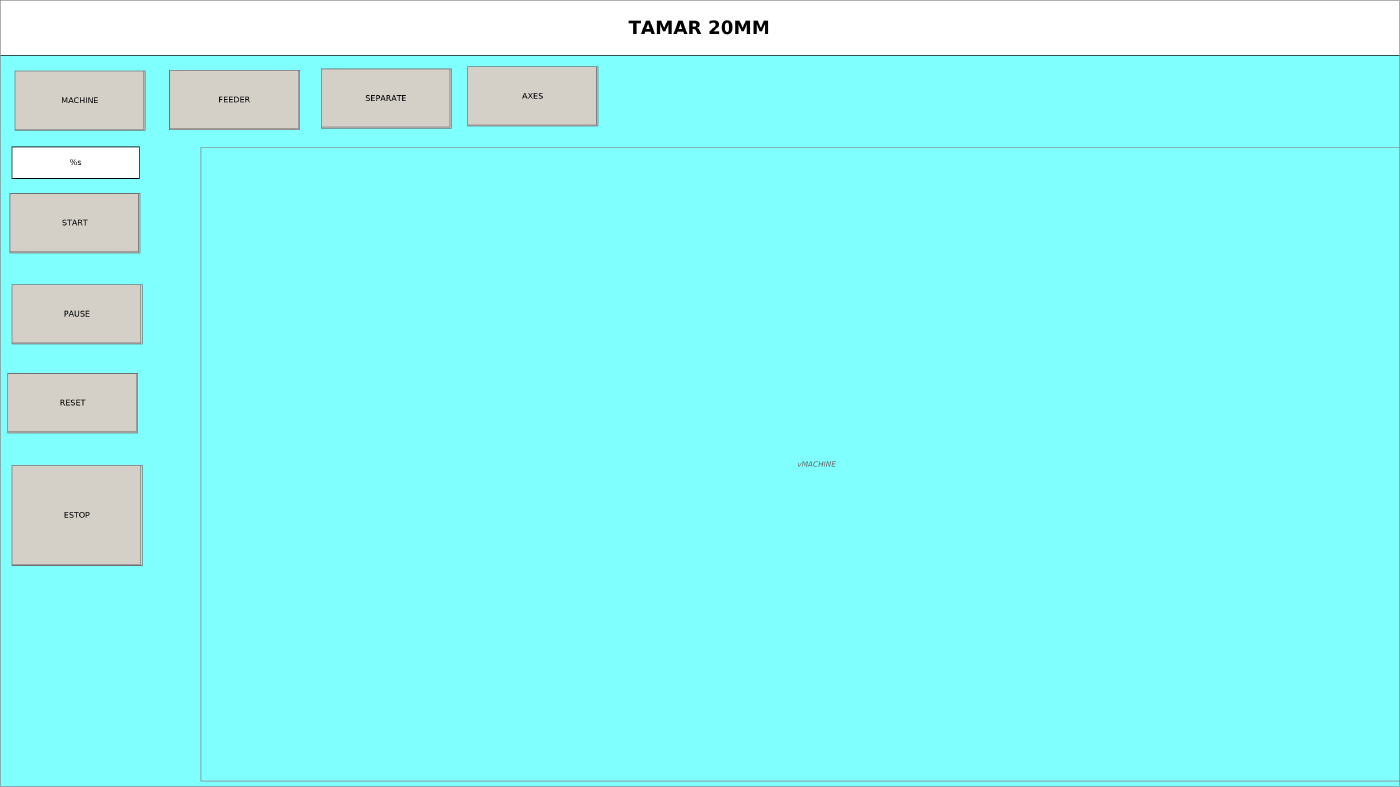
VISUALIZATION vCOMM  // 1920x1080
    Button (13,265 179x82), "START"
        OnMouseClick: execute { bMAIN_START:=TRUE; }
    Rectangle (-3,-1 1924x77), "TAMAR 20MM"
    Button (16,390 179x82), "PAUSE"
    Button (10,512 179x82), "RESET"
        OnMouseClick: execute { bMAIN_RESET:=TRUE; }
    Button (16,638 179x138), "ESTOP"
    Frame (275,202 1690x870)
        shows vMACHINE()
        shows vFEEDER(vFEEDER := fbFEEDER)
        shows vSEPARATE(vSEPARATE1 := fbSEPARATE1, vSEPARATE2 := fbSEPARATE2)
        shows AXES_SCREEN()
    Button (232,96 179x82), "FEEDER"
        OnMouseClick: FrameSelectionChange Selection=SelectedFrame=00e59953-e4a5-4fe1-b8af-e2191fac8d98, Selection=1, GlobSel=AssignType=Directly, SelType=Locally
    Button (20,97 179x82), "MACHINE"
        OnMouseClick: FrameSelectionChange Selection=SelectedFrame=00e59953-e4a5-4fe1-b8af-e2191fac8d98, GlobSel=AssignType=Directly, SelType=Locally
    Button (440,94 179x82), "SEPARATE"
        OnMouseClick: FrameSelectionChange Selection=SelectedFrame=00e59953-e4a5-4fe1-b8af-e2191fac8d98, Selection=2, GlobSel=AssignType=Directly, SelType=Locally
    Rectangle (16,201 175x44), "%s", text variable: sMAIN_STATE
    Button (641,91 179x82), "AXES"
        OnMouseClick: FrameSelectionChange Selection=SelectedFrame=00e59953-e4a5-4fe1-b8af-e2191fac8d98, Selection=3, GlobSel=AssignType=Directly, SelType=Locally
END_VISUALIZATION

(* stored: Version 1.1.0.1, ProductVersion 3.1.4024.12
   Visu vCOMM: Id {da002ba6-ee17-40f4-b476-8d87b46feaa7} *)
